Staubli VAL3: onInsert.pgx

public program onInsert(string& x_sItem[])
  local num l_nDelay
begin
  cls()
  l_nDelay=0
  call use:insertDialog("DELAY [Sec] ",l_nDelay,0,100)
  // give back
  if l_nDelay>0
    if round(l_nDelay)==l_nDelay
      x_sItem=toString("",l_nDelay)
    else
      x_sItem=toString(".2",l_nDelay)
    endIf
  endIf
end
